// TIA Portal V20 export
TYPE "UDT_typeKinCtrl"
   STRUCT
      input : Struct
         bo_estop : Bool;
         bo_enable : Bool;
         bo_reset : Bool;
         bo_home : Bool;
         jogframe : Struct
            "jogX+" : Bool;
            "jogX-" : Bool;
            "jogY+" : Bool;
            "jogY-" : Bool;
            "jogZ+" : Bool;
            "jogZ-" : Bool;
            "jogA+" : Bool;
            "jogA-" : Bool;
            "jogB+" : Bool;
            "jogB-" : Bool;
            "jogC+" : Bool;
            "jogC-" : Bool;
            bo_jogtoposition : Bool;
         END_STRUCT;
         bo_movepathstart : Bool;
         bo_movepathstop : Bool;
         bo_movepathhalt : Bool;
         configuration : Struct
            home { ExternalWritable := 'False'} : Struct
               i16_mode : Array[1..6] of Int;
               r64_homeposition : Array[1..6] of LReal;
            END_STRUCT;
            jogframe : Struct
               targetposition : Struct
                  x : LReal;
                  y : LReal;
                  z : LReal;
                  "a" : LReal;
                  "b" : LReal;
                  c : LReal;
               END_STRUCT;
               dynamics : "LKinCtrl_typeDynamics";   // Specification of the jog dynamics
            END_STRUCT;
         END_STRUCT;
      END_STRUCT;
      output : Struct
         bo_enabled : Bool;
         bo_homed : Bool;
         bo_fault : Bool;
         bo_done : Bool;
         i16_activeCmdNo : Int;
         actualposition : Struct
            x : LReal;
            y : LReal;
            z : LReal;
            "a" : LReal;
            "b" : LReal;
            c : LReal;
         END_STRUCT;
      END_STRUCT;
      inout : Struct
         PathData { S7_SetPoint := 'True'} : "LKinCtrl_typePathData";
      END_STRUCT;
   END_STRUCT;
   // input.configuration.jogframe.dynamics.sPTP.velocityFactor := -1.0;
   // input.configuration.jogframe.dynamics.sPTP.accelerationFactor := -1.0;
   // input.configuration.jogframe.dynamics.sPTP.decelerationFactor := -1.0;
   // input.configuration.jogframe.dynamics.sPTP.jerkFactor := -1.0;
END_TYPE
